# B&R Automation Studio project mappView-Backup
Automation Studio 4.5.4.123 SP

## Configuration X20CPU

### Task classes (Cpu.sw)
```
Cyclic#7:
  Test <- Test.prg
Cyclic#8:
  mappBackup <- mappBackup.mappBackup.prg
  UsbDevice <- USBdevice.UsbDevice.prg
  NetDevice <- NETdevice.NetDevice.prg
Binaries: udbdef, mvLoader, TCData, arsvcreg, sysconf, ashwd, ashwac, asfw, iomap, Role, User, arconfig, OpcUaMap, Config
Libraries: FileIO, runtime, AsBrStr, AsUSB, standard, sys_lib, MpBackup, MpBase, IecCheck, AsBrWStr, astime, asieccon, brsystem, arproject, asarcfg
```

### Hardware
```
X20CP1583 : X20CP1583 v1.5.0.0
  Connector IF2:
    ActivateDevice = 1
  ConfigurationID = Tmp_Backup
  UserPartitionSize = 32
  VolatileGlobalPvSize = 200000
  Cyclic8Stack = 20000
  FileDevice1
  FileDeviceName1 = USER_DEVICE
  FileDevicePath1 = F:/
  FtpUser1
  FtpUsername1 = br
  FtpUserPassword1 = B9fKGuUbjkGCgEptWUpgQ1eJbLeEvMYqPBCteWUIcCw=
  FtpUserSalt1 = wEo/3/qm
  FTPAccessRight1 = 0
  ActivateOpcUa = 1
  OpcUaInformationModels_PV_Version = 1
```

### Config.mpbackupcore - X20CP1583/mappServices/Config.mpbackupcore
```
Element gBackupCore (Type=mpbackupcore)
  Backup:
    AutomaticUpdate = Notify
      DeviceName = USBdevice
```

## Logical view

Binary libraries used (declarations not repeated): operator, runtime, astime, AsIecCon, FileIO, AsBrStr, AsUSB, standard, sys_lib, MpBackup 5.07.1, MpBase, IecCheck, AsBrWStr

### Package Logical/Libraries - Global libraries

- Visualisation Logical/mappView (not shown)

### BackupTypes.typ
```iecst
(*------------------------------------------------------------------------------------------------------------------------------------------------------------------------------------------------------------------------*)
(*Global enumerations*)

TYPE
	bacSTATE :
		( (*Backup managment state machine*)
		BAC_STARTUP,
		BAC_WAIT,
		BAC_CORE,
		BAC_FINISH,
		BAC_GENERATE_NAME,
		BAC_READ_DIR_0,
		BAC_READ_DIR_1,
		BAC_READ_DIR_2,
		BAC_READ_DIR_3,
		BAC_READ_DIR_4,
		BAC_DIR_DELETE,
		BAC_DIR_CREATE,
		BAC_ERROR
		);
END_TYPE

(*------------------------------------------------------------------------------------------------------------------------------------------------------------------------------------------------------------------------*)
(*Global structure*)

TYPE
	bacMAIN : 	STRUCT  (*Backup managment main structure*)
		CMD : bacCMD; (* Command structure *)
		PAR : bacPAR; (* Parameter structure *)
		DAT : bacDAT; (*Data structure*)
		VIS : bacVIS; (*Visualization structure*)
		ERR : bacERR; (* Error structure *)
	END_STRUCT;
	bacCMD : 	STRUCT  (*Backup managment command structure*)
		Backup : BOOL; (*Create a new backup*)
		Restore : BOOL; (*Restore selected backup*)
		Delete : BOOL; (*Delete the selected backaup*)
		GenerateName : BOOL; (*Generate backup name from default name and date*)
		RefreshInfo : BOOL; (*Refresh information for selected backup*)
		RefreshDirectory : BOOL; (*Refresh backup directory names*)
		ErrorReset : BOOL; (*Reset pending errors*)
	END_STRUCT;
	bacPAR : 	STRUCT  (*Backup managment parameter structure*)
		BackupName : STRING[BACKUP_NAME_LENGTH] := 'MyBackup'; (*Name of the variable where the data is stored*)
		DefaultName : STRING[BACKUP_NAME_LENGTH] := 'MyBackup'; (*Name of the variable where the data is stored*)
		DeviceName : STRING[BACKUP_NAME_LENGTH] := 'USB_DEVICE'; (*Device name where the bacipes are stored*)
		UniqueName : STRING[BACKUP_NAME_LENGTH] := 'RestoreInProcessPLC1'; (*Unique name for this PLC to identify if restore was completed*)
		DeviceList : ARRAY[0..4]OF STRING[40]; (*List of all devices*)
		VisuSlotID : USINT; (*ID for connected web connection*)
		ShowMessageBoxOK : BOOL := TRUE;
		ShowMessageBoxError : BOOL := TRUE;
		MpLink : MpComIdentType; (*MpLink from mappBackup*)
	END_STRUCT;
	bacDAT : 	STRUCT  (*Backup managment data structure*)
		CurrentID : STRING[255];
		CurrentVersion : STRING[64];
		RequestedName : STRING[255];
		RequestedID : STRING[255];
		RequestedVersion : STRING[64];
		LastName : STRING[255];
		LastDate : DATE_AND_TIME;
		LastType : MpBackupGenerationTypeEnum;
		BackupNames : ARRAY[0..BACKUP_LIST_NUM]OF STRING[BACKUP_NAME_LENGTH];
		BackupNum : USINT;
		Status : WSTRING[200]; (*Shows the result of the last command*)
	END_STRUCT;
	bacVIS : 	STRUCT  (*Backup managment visualization structure*)
		DeviceList : ARRAY[0..4]OF STRING[80]; (* Device name *)
		BackupNames : ARRAY[0..BACKUP_LIST_NUM]OF STRING[BACKUP_VIS_LENGTH];
		EnableCommand : BOOL;
		EnableDelete : BOOL;
		ShowMessageBoxOK : BOOL;
		ShowMessageBoxError : BOOL;
	END_STRUCT;
	bacERR : 	STRUCT  (*Backup managment error structure*)
		Text : WSTRING[200]; (* Error text *)
		No : DINT; (* Error number *)
		State : bacSTATE; (* Error step *)
	END_STRUCT;
END_TYPE
```

### BackupVariables.var
```iecst
VAR CONSTANT
	BACKUP_DEVICE_LIST : ARRAY[0..4] OF STRING[40] := ['USB_DEVICE','NET_DEVICE',3('')]; (*List of predefined devices *)
	BACKUP_LIST_NUM : UINT := 20; (*Maximum number of backups*)
	BACKUP_NAME_LENGTH : UINT := 100; (*Maximum length for a backup name*)
	BACKUP_VIS_LENGTH : UINT := 300; (*Make this BACKUP_NAME_LENGTH  x3*)
END_VAR
VAR
	BACKUP_DIRECTORY : STRING[200]; (*Directory for backups*)
	Backup_01 : bacMAIN; (*Backup management main structure*)
END_VAR
```

### Program Logical/mappBackup/mappBackup (IEC) - Sample for all AsUSB-Library-Functions

#### Backup.st - Cyclic code
```iecst
// ----------------------------------------------------------------------------------------
//	Function:	Software management for B&R PLCs
//  Version:	0.1
//	Changed:	11.11.2019
//	Error numbers:
//	50000		Backup name is empty
//	50001		Device name is empty
//	50010		Maximum number of backup names reached
//	50011		Backup name length exceeds maximum size
//	50020		Backup name already exists
// ----------------------------------------------------------------------------------------

PROGRAM _INIT
	// ----------------------------------------------------------------------------------------
	Backup_01.PAR.MpLink := gBackupCore;				// Link to mappBackup configuration

	// ----------------------------------------------------------------------------------------
	brsmemcpy(ADR(Backup_01.PAR.DeviceList), ADR(BACKUP_DEVICE_LIST), SIZEOF(BACKUP_DEVICE_LIST));
	Backup_01.DAT.Status := "Waiting...";

	MpBackupCore_0.MpLink := ADR(Backup_01.PAR.MpLink);
	MpBackupCore_0.Name := ADR(BackupName);
	MpBackupCore_0.DeviceName := ADR(DeviceName);

END_PROGRAM

PROGRAM _CYCLIC
	// --------------------------------------------------------------------------------------------------------------------
	// Cyclic function call
	MpBackupCore_0.Enable := 1;
	MpBackupCore_0();

	// ------------------------------------------------------------------------------------------------
	// Generate device name list
	brsmemset(ADR(Backup_01.VIS.DeviceList), 0, SIZEOF(Backup_01.VIS.DeviceList));
	FOR idx := 0 TO SIZEOF(Backup_01.VIS.DeviceList)/SIZEOF(Backup_01.VIS.DeviceList[0]) - 1 DO
		IF (Backup_01.PAR.DeviceList[idx] <> '') THEN
			String2DataProvider(ADR(Backup_01.PAR.DeviceList[idx]), ADR(Backup_01.VIS.DeviceList[idx]));
		END_IF
	END_FOR;

	// ------------------------------------------------------------------------------------------------
	// Generate backup name list
	brsmemset(ADR(Backup_01.VIS.BackupNames), 0, SIZEOF(Backup_01.VIS.BackupNames));
	IF(Backup_01.DAT.BackupNum > 0) THEN
		FOR idx := 0 TO Backup_01.DAT.BackupNum - 1 DO
			IF (Backup_01.DAT.BackupNames[idx] <> '') THEN
				String2DataProvider(ADR(Backup_01.DAT.BackupNames[idx]), ADR(Backup_01.VIS.BackupNames[idx]));
			END_IF
		END_FOR;
	END_IF

	// ------------------------------------------------------------------------------------------------
	// Enable/Disable visualization elements
	IF(bac_state <> BAC_WAIT) THEN
		Backup_01.VIS.EnableCommand := FALSE;
	ELSE
		Backup_01.VIS.EnableCommand := TRUE;
	END_IF
	IF(Backup_01.DAT.BackupNum = 0) THEN
		Backup_01.VIS.EnableDelete := FALSE;
	ELSE
		Backup_01.VIS.EnableDelete := TRUE;
	END_IF

	//**************************************************************************************************
	// Backup managment state machine
	//**************************************************************************************************
	CASE bac_state OF
		//**********************************************************************************************
		// Wait for USB and network connection to startup
		//**********************************************************************************************
		BAC_STARTUP:
			Backup_01.DAT.Status := "Waiting for USB and network connections to startup";
			StartupDelay(IN := 1, PT := DELAY_STARTUP);
			IF (StartupDelay.Q) THEN
				bac_state := BAC_WAIT;
			END_IF
		//**********************************************************************************************
		// Wait for command
		//**********************************************************************************************
		BAC_WAIT:
			// ----------------------------------------------------------------------------------------
			// Make sure device name is not empty
			IF ((Backup_01.CMD.Backup = TRUE OR Backup_01.CMD.Restore = TRUE OR Backup_01.CMD.Delete = TRUE OR Backup_01.CMD.RefreshDirectory = TRUE OR Backup_01.CMD.RefreshInfo = TRUE) AND Backup_01.PAR.DeviceName = '') THEN
				bac_state := CreateError(ADR(Backup_01), ERR_BAC_NAME_IS_EMPTY, "Device name is empty", bac_state);
				RETURN;
			ELSE
				// Freeze device name
				DeviceName := Backup_01.PAR.DeviceName;
			END_IF

			// ----------------------------------------------------------------------------------------
			// Make sure backup name is not empty
			IF ((Backup_01.CMD.Backup = TRUE OR Backup_01.CMD.Restore = TRUE OR Backup_01.CMD.Delete = TRUE OR Backup_01.CMD.RefreshInfo = TRUE) AND Backup_01.PAR.BackupName = '') THEN
				bac_state := CreateError(ADR(Backup_01), ERR_BAC_DEVICE_IS_EMPTY, "Backup name is empty", bac_state);
				RETURN;
			ELSE
				// Freeze backup name
				BackupName := Backup_01.PAR.BackupName;
			END_IF

			// ------------------------------------------------------------------------------------------------
			// Track device name change
			IF (brsstrcmp(ADR(DeviceNameOld), ADR(DeviceName)) <> 0) THEN
				Backup_01.CMD.RefreshDirectory	:= 1;
			END_IF
			DeviceNameOld := DeviceName;

			// ----------------------------------------------------------------------------------------
			// Command restore backup
			IF (Backup_01.CMD.Restore = TRUE) THEN
				// Show current state
				tmpWStr1 := "Restoring backup...";
				bac_state := BAC_DIR_CREATE;
			// ----------------------------------------------------------------------------------------
			// Command create backup
			ELSIF (Backup_01.CMD.Backup = TRUE) THEN
				// Make sure that backup name does not already exist
				IF(Backup_01.DAT.BackupNum > 0) THEN
					FOR idx:=0 TO Backup_01.DAT.BackupNum - 1 DO
						IF(brsstrcmp(ADR(BackupName), ADR(Backup_01.DAT.BackupNames[idx])) = 0) THEN
							bac_state := CreateError(ADR(Backup_01), ERR_BAC_NAME_EXISTS, "Backup name already exists", bac_state);
							RETURN;
						END_IF
					END_FOR;
				END_IF

				// Show current state
				tmpWStr1 := "Creating backup...";
				bac_state := BAC_CORE;
			// ----------------------------------------------------------------------------------------
			// Command delete backup
			ELSIF (Backup_01.CMD.Delete = TRUE) THEN
				// Show current state
				tmpWStr1 := "Deleting backup...";
				bac_state := BAC_DIR_DELETE;
			// ----------------------------------------------------------------------------------------
			// Command refresh backup information
			ELSIF (Backup_01.CMD.RefreshInfo = TRUE) THEN
				// Show current state
				tmpWStr1 := "Refreshing backup information...";
				bac_state := BAC_CORE;
			// ----------------------------------------------------------------------------------------
			// Command refresh device information
			ELSIF (Backup_01.CMD.RefreshDirectory = TRUE) THEN
				// Show current state
				tmpWStr1 := "Refreshing direct ory information...";
				DeviceIdx := 0;
				found_restore_dir := FALSE;
				DeviceName := Backup_01.PAR.DeviceName;
				bac_state := BAC_READ_DIR_0;
			// ----------------------------------------------------------------------------------------
			// Command generate backup name
			ELSIF (Backup_01.CMD.GenerateName = TRUE) THEN
				// Generate backup name
				bac_state := BAC_GENERATE_NAME;
			// ----------------------------------------------------------------------------------------
			// Command reset error
			ELSIF (Backup_01.CMD.ErrorReset = TRUE) THEN
				// Generate backup name
				bac_state := BAC_ERROR;
			END_IF

			animation := 0;
			MpBackupCore_0.ErrorReset := FALSE;
		//**********************************************************************************************
		// Generate backup name
		//**********************************************************************************************
		BAC_GENERATE_NAME:
			// Generate backup name using default name and date
			Backup_01.PAR.BackupName := Backup_01.PAR.DefaultName;
			RTC_gettime(ADR(rtc_gettime));
			brsstrcat(ADR(Backup_01.PAR.BackupName), ADR('_D'));
			IF(rtc_gettime.day < 10) THEN
				brsstrcat(ADR(Backup_01.PAR.BackupName), ADR('0'));
			END_IF
			brsitoa(rtc_gettime.day, ADR(tmpStr1));
			brsstrcat(ADR(Backup_01.PAR.BackupName), ADR(tmpStr1));
			brsitoa(rtc_gettime.day, ADR(tmpStr1));
			brsstrcat(ADR(Backup_01.PAR.BackupName), ADR('_M'));
			IF(rtc_gettime.month < 10) THEN
				brsstrcat(ADR(Backup_01.PAR.BackupName), ADR('0'));
			END_IF
			brsitoa(rtc_gettime.month, ADR(tmpStr1));
			brsstrcat(ADR(Backup_01.PAR.BackupName), ADR(tmpStr1));
			brsstrcat(ADR(Backup_01.PAR.BackupName), ADR('_Y'));
			brsitoa(rtc_gettime.year, ADR(tmpStr1));
			brsstrcat(ADR(Backup_01.PAR.BackupName), ADR(tmpStr1));
			brsstrcat(ADR(Backup_01.PAR.BackupName), ADR('_h'));
			IF(rtc_gettime.hour < 10) THEN
				brsstrcat(ADR(Backup_01.PAR.BackupName), ADR('0'));
			END_IF
			brsitoa(rtc_gettime.hour, ADR(tmpStr1));
			brsstrcat(ADR(Backup_01.PAR.BackupName), ADR(tmpStr1));
			brsstrcat(ADR(Backup_01.PAR.BackupName), ADR('_m'));
			IF(rtc_gettime.minute < 10) THEN
				brsstrcat(ADR(Backup_01.PAR.BackupName), ADR('0'));
			END_IF
			brsitoa(rtc_gettime.minute, ADR(tmpStr1));
			brsstrcat(ADR(Backup_01.PAR.BackupName), ADR(tmpStr1));
			brsstrcat(ADR(Backup_01.PAR.BackupName), ADR('_s'));
			IF(rtc_gettime.second < 10) THEN
				brsstrcat(ADR(Backup_01.PAR.BackupName), ADR('0'));
			END_IF
			brsitoa(rtc_gettime.second, ADR(tmpStr1));
			brsstrcat(ADR(Backup_01.PAR.BackupName), ADR(tmpStr1));

			Backup_01.CMD.GenerateName := FALSE;
			bac_state := BAC_WAIT;
		// --------------------------------------------------------------------------------------------------------------------
		// Core function call
		// --------------------------------------------------------------------------------------------------------------------
		BAC_CORE:
			// ------------------------------------------------------------------------------------------------
			// Main backup function call
			animation := WorkingStatus(ADR(Backup_01), ADR(tmpWStr1), animation);

			// ----------------------------------------------------------------------------------------
			// OK
			IF (MpBackupCore_0.CommandDone AND NOT MpBackupCore_0.Error) THEN
				IF(Backup_01.CMD.RefreshInfo OR Backup_01.CMD.Restore) THEN
					bac_state := BAC_FINISH;
				ELSE
					bac_state := BAC_READ_DIR_0;
				END_IF
				// ----------------------------------------------------------------------------------------
			// Error
			ELSIF (MpBackupCore_0.Error) THEN
				// ----------------------------------------------------------------------------------------
				// Generate error message depending on initial command
				IF (Backup_01.CMD.Backup) THEN
					IF(MpBackupCore_0.StatusID =  mpBACKUP_ERR_CREATE_FAILED) THEN
						tmpWStr1 := "Backup name already exists";
					ELSE
						tmpWStr1 := "Error trying to backup data";
					END_IF
				ELSIF (Backup_01.CMD.Restore) THEN
					IF(MpBackupCore_0.StatusID =  mpBACKUP_ERR_INSTALL_FAILED) THEN
						tmpWStr1 := "Can not find backup name";
					ELSE
						tmpWStr1 := "Error trying to restore data";
					END_IF
				ELSIF (Backup_01.CMD.RefreshInfo) THEN
					IF(MpBackupCore_0.StatusID =  mpBACKUP_ERR_REQUEST_INFO_FAILED) THEN
						bac_state := BAC_FINISH;
						RETURN;
					ELSE
						tmpWStr1 := "Error trying to refresh backup information";
					END_IF
				END_IF
				bac_state := CreateError(ADR(Backup_01), MpBackupCore_0.StatusID, tmpWStr1, bac_state);
			END_IF
		//**********************************************************************************************
		// Finish command
		//**********************************************************************************************
		BAC_FINISH:
			// ----------------------------------------------------------------------------------------
			// Comand backup
			IF (Backup_01.CMD.Backup) THEN
				// Reset command, set status and show message box
				Backup_01.DAT.Status := "Backup completed";
				IF(Backup_01.PAR.ShowMessageBoxOK) THEN
					Backup_01.VIS.ShowMessageBoxOK := TRUE;
				END_IF
			// ----------------------------------------------------------------------------------------
			// Comand restore
			ELSIF (Backup_01.CMD.Restore) THEN
				// Reset command, set status, return to wait state
				Backup_01.DAT.Status := "Restore backup completed";
			// ----------------------------------------------------------------------------------------
			// Comand delete
			ELSIF (Backup_01.CMD.Delete) THEN
				// Reset command, set status, return to wait state
				Backup_01.DAT.Status := "Deleted backup";
				IF(Backup_01.PAR.ShowMessageBoxOK) THEN
					Backup_01.VIS.ShowMessageBoxOK := TRUE;
				END_IF
			// ----------------------------------------------------------------------------------------
			// Comand refresh backup names
			ELSIF (Backup_01.CMD.RefreshDirectory) THEN
				// Show error message if there are oversized items
				IF(found_restore_dir) THEN
					// Reset command, set status, return to wait state
					found_restore_dir := FALSE;
					Backup_01.DAT.Status := "Restore backup complete";
					IF(Backup_01.PAR.ShowMessageBoxOK) THEN
						Backup_01.VIS.ShowMessageBoxOK := TRUE;
					END_IF
				ELSE
					Backup_01.DAT.Status := "Refreshed backup names";
				END_IF
			// ----------------------------------------------------------------------------------------
			// Comand refresh backup information
			ELSIF (Backup_01.CMD.RefreshInfo) THEN
				// Directory does not contain a PLC backup
				IF(MpBackupCore_0.StatusID =  mpBACKUP_ERR_REQUEST_INFO_FAILED) THEN
					Backup_01.DAT.Status := "Can not find directory or backup information";
				ELSE
					Backup_01.DAT.Status := "Refreshed backup information";
				END_IF
			END_IF
			// Set status, return to wait state
			brsmemset(ADR(Backup_01.CMD), 0, SIZEOF(Backup_01.CMD));
			MpBackupCore_0.ErrorReset := TRUE;
			MpBackupCore_0();
			MpBackupCore_0.ErrorReset := FALSE;
			bac_state := BAC_WAIT;
		//**********************************************************************************************
		// Read directory information
		//**********************************************************************************************
		BAC_READ_DIR_0:
			// Show current state
			animation := WorkingStatus(ADR(Backup_01), ADR(tmpWStr1), animation);
			// Clear all entrys, reset mappBackup function block
			brsmemset(ADR(Backup_01.DAT), 0, SIZEOF(Backup_01.DAT));
			Backup_01.DAT.BackupNum := 0;
			has_oversized_items := FALSE;

			// ----------------------------------------------------------------------------------------
			// Reset mappBackup function block
			MpBackupCore_0.Enable := 0;
			MpBackupCore_0();
			// ----------------------------------------------------------------------------------------
			// Set values and get device dir
			DInfo.enable 	:= 1;
			DInfo.pDevice	:= ADR(DeviceName);
			DInfo();

			// ----------------------------------------------------------------------------------------
			// OK
			IF (DInfo.status = OK) THEN
				first_boot := FALSE;
				bac_state := BAC_READ_DIR_1;
			ELSIF (DInfo.status = fiERR_DEVICE_MANAGER) THEN
				// On first boot skip devices that are not available
				IF (first_boot) THEN
					DeviceIdx := DeviceIdx + 1;
					IF(Backup_01.PAR.DeviceList[DeviceIdx] <> '') THEN
						brsstrcpy(ADR(DeviceName), ADR(Backup_01.PAR.DeviceList[DeviceIdx]));
						brsstrcpy(ADR(DeviceNameOld), ADR(Backup_01.PAR.DeviceList[DeviceIdx]));
						brsstrcpy(ADR(Backup_01.PAR.DeviceName), ADR(Backup_01.PAR.DeviceList[DeviceIdx]));
					ELSE
						// Set status, return to wait state
						brsmemset(ADR(Backup_01.CMD), 0, SIZEOF(Backup_01.CMD));
						first_boot := FALSE;
						bac_state := BAC_WAIT;
					END_IF
				// Create error message when file device is not available
				ELSE
					tmpWStr1 := "File device ";
					brwcsconv(ADR(tmpWStr2), ADR(DeviceName), brwU8toUC);
					brwcscat(ADR(tmpWStr1), ADR(tmpWStr2));
					brwcscat(ADR(tmpWStr1), ADR(" is unavailable"));
					bac_state := CreateError(ADR(Backup_01), DInfo.status, tmpWStr1, bac_state);
				END_IF
			// Error
			ELSIF (DInfo.status <> ERR_FUB_BUSY) THEN
				first_boot := FALSE;
				bac_state := CreateError(ADR(Backup_01), DInfo.status, "Error dir info", bac_state);
			END_IF
		//**********************************************************************************************
		// Open directory
		//**********************************************************************************************
		BAC_READ_DIR_1:
			// Show current state
			animation := WorkingStatus(ADR(Backup_01), ADR(tmpWStr1), animation);

			DOpen.enable 	:= 1;
			DOpen.pDevice	:= ADR(DeviceName);
			DOpen.pName 	:= ADR(BACKUP_DIRECTORY);
			DOpen();

			// ----------------------------------------------------------------------------------------
			// OK
			IF (DOpen.status = OK) THEN
				bac_state := BAC_READ_DIR_2;
				// Error
			ELSIF (DOpen.status <> ERR_FUB_BUSY) THEN
				bac_state := CreateError(ADR(Backup_01), DOpen.status, "Error dir open", bac_state);
			END_IF;
		//**********************************************************************************************
		// Read file directory information
		//**********************************************************************************************
		BAC_READ_DIR_2:
			// Show current state
			animation := WorkingStatus(ADR(Backup_01), ADR(tmpWStr1), animation);

			DRead.enable 	:= 1;
			DRead.ident		:= DOpen.ident;
			DRead.pData 	:= ADR(lDirReadData);
			DRead.data_len 	:= SIZEOF(lDirReadData);
			DRead();

			// ----------------------------------------------------------------------------------------
			// OK
			IF (DRead.status = OK AND lDirReadData.Mode = fiDIRECTORY AND brsstrcmp(ADR(lDirReadData.Filename), ADR('.')) <> 0 AND brsstrcmp(ADR(lDirReadData.Filename), ADR('..')) <> 0 AND brsstrcmp(ADR(lDirReadData.Filename), ADR('System Volume Information')) <> 0) THEN
				// Make sure file name does not exceed maximum string size
				IF (brsstrlen(ADR(lDirReadData.Filename)) < BACKUP_NAME_LENGTH) THEN
					// Copy dir info to string
					brsmemset(ADR(tmpStr1), 0, SIZEOF(tmpStr1));
					brsstrcpy(ADR(tmpStr1), ADR(lDirReadData.Filename));
					// Found restore directory
					IF(brsstrcmp(ADR(Backup_01.PAR.UniqueName), ADR(tmpStr1)) = 0) THEN
						found_restore_dir := TRUE;
					ELSE
						// ------------------------------------------------------------------------------------
						// Verify that we still have space in list
						IF (Backup_01.DAT.BackupNum <= BACKUP_LIST_NUM) THEN
							InsertRecName(ADR(Backup_01), tmpStr1);
							// Error
						ELSE
							bac_state := CreateError(ADR(Backup_01), ERR_BAC_MAX_NUM, "Maximum number of backups reached", bac_state);
						END_IF
					END_IF
				ELSE
					has_oversized_items := TRUE;
				END_IF
			// Last entry reached
			ELSIF (DRead.status = fiERR_NO_MORE_ENTRIES) THEN
				bac_state := BAC_READ_DIR_3;
			// Error
			ELSIF (DRead.status <> ERR_FUB_BUSY AND DRead.status <> OK) THEN
				bac_state := CreateError(ADR(Backup_01), DRead.status, "Error backup list read", bac_state);
			END_IF
		//**********************************************************************************************
		// Close directory information
		//**********************************************************************************************
		BAC_READ_DIR_3:
			// Show current state
			animation := WorkingStatus(ADR(Backup_01), ADR(tmpWStr1), animation);

			DClose.enable 	:= 1;
			DClose.ident	:= DOpen.ident;
			DClose();

			// ----------------------------------------------------------------------------------------
			// OK
			IF (DClose.status = OK) THEN
				// Delete restore flag directory
				IF(found_restore_dir) THEN
					BackupName := Backup_01.PAR.UniqueName;
					bac_state := BAC_DIR_DELETE;
				// Finish directory reading
				ELSE
					bac_state := BAC_READ_DIR_4;
				END_IF
			// Error
			ELSIF (DClose.status <> ERR_FUB_BUSY) THEN
				bac_state := CreateError(ADR(Backup_01), DClose.status, "Error dir close", bac_state);
			END_IF
		//**********************************************************************************************
		// Finish directory information
		//**********************************************************************************************
		BAC_READ_DIR_4:
			// Show error message if there are oversized items
			IF(has_oversized_items) THEN
				bac_state := CreateError(ADR(Backup_01), ERR_BAC_NAME_LENGTH, "One or more backup names exceeds maximum length", bac_state);
			ELSE
				// Get information from first entry
				IF(Backup_01.DAT.BackupNum > 0) THEN
					BackupName := Backup_01.DAT.BackupNames[0];
					Backup_01.CMD.RefreshInfo := TRUE;
					bac_state := BAC_CORE;
				ELSE
					bac_state := BAC_FINISH;
				END_IF
			END_IF
		//**********************************************************************************************
		// Delete selected directory
		//**********************************************************************************************
		BAC_DIR_DELETE:
			// Show current state
			animation := WorkingStatus(ADR(Backup_01), ADR("Deleting backup..."), animation);

			// ----------------------------------------------------------------------------------------
			// Initialize directory delete structure
			DDelete.enable	:= 1;
			DDelete.pDevice := ADR(DeviceName);
			DDelete.pName 	:= ADR(BackupName);
			DDelete();

			// ----------------------------------------------------------------------------------------
			// OK
			IF (DDelete.status = OK) THEN
				// Deleted restore directory
				IF(found_restore_dir) THEN
					bac_state := BAC_READ_DIR_4;
				// Deleted standard backup directory
				ELSE
					// Show status and return to wait state
					Backup_01.DAT.Status := "Deleted backup";
					bac_state := BAC_READ_DIR_0;
				END_IF
			// Error
			ELSIF (DDelete.status <> ERR_FUB_BUSY) THEN
				IF(DDelete.status = fiERR_DIR_NOT_EXIST) THEN
					bac_state := CreateError(ADR(Backup_01), DDelete.status, "Can not find backup directory", bac_state);
				ELSE
					bac_state := CreateError(ADR(Backup_01), DDelete.status, "Error deleting backup", bac_state);
				END_IF
			END_IF
		//**********************************************************************************************
		// Create selected directory
		//**********************************************************************************************
		BAC_DIR_CREATE:
			// Show current state
			animation := WorkingStatus(ADR(Backup_01), ADR(tmpWStr1), animation);

			// ----------------------------------------------------------------------------------------
			// Initialize directory delete structure
			DCreate.enable	:= 1;
			DCreate.pDevice := ADR(DeviceName);
			DCreate.pName 	:= ADR(Backup_01.PAR.UniqueName);
			DCreate();

			// ----------------------------------------------------------------------------------------
			// OK
			IF (DCreate.status = OK OR DCreate.status = fiERR_DIR_ALREADY_EXIST) THEN
				// Start restoring backup
				bac_state := BAC_CORE;
			// Error
			ELSIF (DCreate.status <> ERR_FUB_BUSY) THEN
				bac_state := CreateError(ADR(Backup_01), DCreate.status, "Could not create restore flag directory", bac_state);
			END_IF
		// --------------------------------------------------------------------------------------------------------------------
		// Error
		// --------------------------------------------------------------------------------------------------------------------
		BAC_ERROR:
			Backup_01.DAT.Status := "Acknowledge error to trigger new command";

			// Make sure we dont exceed maximum number of web clients
			IF(Backup_01.PAR.ShowMessageBoxError) THEN
				Backup_01.VIS.ShowMessageBoxError := TRUE;
			END_IF
			// --------------------------------------------------------------------------------------------------------------------
			// Return to idle state
			IF (Backup_01.CMD.ErrorReset) THEN
				// Reset function blocks
				MpBackupCore_0.ErrorReset := TRUE;
				MpBackupCore_0();
				MpBackupCore_0.ErrorReset := FALSE;

				// Reset error structure
				brsmemset(ADR(Backup_01.ERR), 0, SIZEOF(Backup_01.ERR));
				Backup_01.DAT.Status := "";
				Backup_01.VIS.ShowMessageBoxError := FALSE;
				bac_state := BAC_WAIT;
			END_IF;
			brsmemset(ADR(Backup_01.CMD), 0, SIZEOF(Backup_01.CMD));
	END_CASE

	// --------------------------------------------------------------------------------------------------------------------
	// Cyclic function call
	MpBackupCore_0.Enable := 1;
	MpBackupCore_0.Create := Backup_01.CMD.Backup;
	MpBackupCore_0.Install := Backup_01.CMD.Restore;
	MpBackupCore_0.RequestInfo := Backup_01.CMD.RefreshInfo;
	MpBackupCore_0();

	Backup_01.DAT.CurrentID := MpBackupCore_0.Info.Project.Current.ConfigurationID;
	Backup_01.DAT.CurrentVersion := MpBackupCore_0.Info.Project.Current.ConfigurationVersion;
	Backup_01.DAT.RequestedName := MpBackupCore_0.Info.Project.Requested.Name;
	Backup_01.DAT.RequestedID := MpBackupCore_0.Info.Project.Requested.ConfigurationID;
	Backup_01.DAT.RequestedVersion := MpBackupCore_0.Info.Project.Requested.ConfigurationVersion;
	Backup_01.DAT.LastName := MpBackupCore_0.Info.LastBackup.Name;
	Backup_01.DAT.LastDate := MpBackupCore_0.Info.LastBackup.DateTime;
	Backup_01.DAT.LastType := MpBackupCore_0.Info.LastBackup.GenerationType;

END_PROGRAM

PROGRAM _EXIT
	MpBackupCore_0.Enable := 0;
	MpBackupCore_0();
END_PROGRAM
```

#### Backup.var - Data for read_data Task
```iecst
(*------------------------------------------------------------------------------------------------------------------------------------------------------------------------------------------------------------------------*)
(*Local constants*)
VAR CONSTANT
	OK : USINT := 0; (*Constant for status OK *)
END_VAR
VAR
	DELAY_STARTUP : UINT := 1000; (*Delay startup to give USB and network connections time to start up*)
END_VAR
(*----------------------------------------------------------------------------------------------------------------------------------------------------------------------------------------------------------------------------------------------------------------------*)
(*Local variables*)
VAR
	bac_state : bacSTATE := BAC_STARTUP; (*Main step index *)
	first_boot : BOOL := TRUE; (*Flag for first boot up, run some special code*)
	animation : UDINT := 0; (*Animation for working status	*)
	tmpWStr1 : WSTRING[200]; (*Temporary unicode string variable *)
	tmpWStr2 : WSTRING[200]; (*Temporary unicode string variable *)
	tmpStr1 : STRING[100]; (*Temporary string variable *)
	BackupName : STRING[BACKUP_NAME_LENGTH]; (*Local backup name*)
	DeviceNameOld : STRING[100]; (*Local device name*)
	DeviceName : STRING[100]; (*Local device name*)
	DeviceIdx : USINT;
	idx : UINT; (*Counter variable*)
	rtc_gettime : RTCtime_typ; (*Time and date*)
	lDirReadData : fiDIR_READ_EX_DATA; (*File and directory information*)
	has_oversized_items : BOOL; (*Flag for oversized backup names*)
	found_restore_dir : BOOL; (*Flag for directory for the restpre process*)
END_VAR
(*----------------------------------------------------------------------------------------------------------------------------------------------------------------------------------------------------------------------------------------------------------------------*)
(*Local functions*)
VAR
	MpBackupCore_0 : MpBackupCore; (*mappBackup function block*)
	DInfo : DirInfo; (*Directory information*)
	DOpen : DirOpen; (*Start reading directories*)
	DRead : DirReadEx; (*Read directories*)
	DClose : DirClose; (*Finish reading directories*)
	DDelete : DirDeleteEx; (*Delete directory*)
	DCreate : DirCreate; (*Finish reading directories*)
	StartupDelay : TON_10ms; (*Delay startup timer*)
END_VAR
(*----------------------------------------------------------------------------------------------------------------------------------------------------------------------------------------------------------------------------------------------------------------------*)
(*Local errors*)
VAR
	ERR_BAC_NAME_IS_EMPTY : DINT := 50000; (*Backup name is empty*)
	ERR_BAC_DEVICE_IS_EMPTY : DINT := 50001; (*Device name is empty*)
	ERR_BAC_MAX_NUM : DINT := 50010; (*Maximum number of backup names reached*)
	ERR_BAC_NAME_LENGTH : DINT := 50011; (*Backup name length exceeds maximum size*)
	ERR_BAC_NAME_EXISTS : DINT := 50020; (*Backup name already exists*)
END_VAR
```

#### LocalFunctions.fun
```iecst
FUNCTION String2DataProvider : BOOL
	VAR_INPUT
		SourceString : UDINT;
		TargetString : UDINT;
	END_VAR
END_FUNCTION

FUNCTION WorkingStatus : UDINT
	VAR_INPUT
		BACKUP : REFERENCE TO bacMAIN;
		str : UDINT;
		animation : UDINT;
	END_VAR
	VAR
		counter : UDINT;
		tmpStr : STRING[20];
		tmpWStr : WSTRING[20];
	END_VAR
END_FUNCTION

FUNCTION CreateError : bacSTATE
	VAR_INPUT
		BACKUP : REFERENCE TO bacMAIN;
		No : DINT;
		Text : WSTRING[200];
		State : bacSTATE;
	END_VAR
END_FUNCTION

FUNCTION InsertRecName : BOOL
	VAR_INPUT
		BAC : REFERENCE TO bacMAIN;
		new_name : STRING[BACKUP_NAME_LENGTH];
	END_VAR
	VAR
		idx : DINT;
		idy : DINT;
		lSort : DINT;
	END_VAR
END_FUNCTION
```

#### LocalFunctions.st
```iecst
//******************************************************************************************************
// Create mappView data provider string
//******************************************************************************************************
FUNCTION String2DataProvider
	brsstrcpy(TargetString, ADR('{"value":"'));
	brsstrcat(TargetString, SourceString);
	brsstrcat(TargetString, ADR('","text":"'));
	brsstrcat(TargetString, SourceString);
	brsstrcat(TargetString, ADR('"}'));
	String2DataProvider := TRUE;
END_FUNCTION

//******************************************************************************************************
// Create error
//******************************************************************************************************
FUNCTION CreateError
	BACKUP.ERR.No := No;
	BACKUP.ERR.State := State;
	BACKUP.ERR.Text := Text;
	CreateError := BAC_ERROR;
END_FUNCTION

//******************************************************************************************************
// Working status
//******************************************************************************************************
FUNCTION WorkingStatus
	animation := animation+1;

	// Get one second counter
	counter := animation;
	WHILE counter >= 100 DO
		counter := counter - 100;
	END_WHILE;

	IF (counter = 99) THEN
		counter := 0;
	END_IF

	// Add counter to output string
	brsmemset(ADR(BACKUP.DAT.Status), 0, SIZEOF(BACKUP.DAT.Status));
	brwcscpy(ADR(BACKUP.DAT.Status), str);
	brwcscat(ADR(BACKUP.DAT.Status), ADR(" "));
	brsitoa(animation/100, ADR(tmpStr));
	brwcsconv(ADR(tmpWStr), ADR(tmpStr), brwU8toUC);
	brwcscat(ADR(BACKUP.DAT.Status), ADR(tmpWStr));
	brwcscat(ADR(BACKUP.DAT.Status), ADR("s "));

	// Add rotating element to output string
	CASE(counter) OF
		0..24	: brwcscat(ADR(BACKUP.DAT.Status), ADR("/"));
		25..49	: brwcscat(ADR(BACKUP.DAT.Status), ADR("-"));
		50..74	: brwcscat(ADR(BACKUP.DAT.Status), ADR("\"));
		75..99	: brwcscat(ADR(BACKUP.DAT.Status), ADR("|"));
	END_CASE;
	WorkingStatus := animation;
END_FUNCTION

//******************************************************************************************************
// Fill in new directory name
//******************************************************************************************************
FUNCTION InsertRecName
	// Set up start values for iteration
	IF (BAC.DAT.BackupNum <> 0) THEN
		idy := BAC.DAT.BackupNum - 1;
	END_IF
	idx := idy;

	// Start iteration	search
	WHILE (idy > 1) DO
		// Check current entry
		lSort := brsstrcmp(ADR(new_name), ADR(BAC.DAT.BackupNames[idy]));
		// Solve new search range
		IF (idy MOD 2 = 0) THEN
			idy := idy / 2;
		ELSE
			idy := idy / 2 + 1;
		END_IF
		// New range is lower or higher than current
		IF (lSort > 0) THEN
			idx := idx + idy;
			IF (idx > UINT_TO_INT(BAC.DAT.BackupNum)) THEN
				idx := BAC.DAT.BackupNum;
			END_IF
		ELSE
			idx := idx - idy;
			IF (idx < 1) THEN
				idx := 1;
			END_IF
		END_IF
	END_WHILE;

	// New entry is this, next or previous
	lSort := brsstrcmp(ADR(new_name), ADR(BAC.DAT.BackupNames[idx]));
	IF (lSort > 0 AND idx <> UINT_TO_INT(BAC.DAT.BackupNum)) THEN
		idx := idx +1;
	ELSIF (idx > 0) THEN
		lSort := brsstrcmp(ADR(new_name), ADR(BAC.DAT.BackupNames[idx-1]));
		IF (lSort < 0) THEN
			idx := idx - 1;
		END_IF
	END_IF

	// Move all data entrys backwards and fill in new entry
	IF(idx < BACKUP_LIST_NUM) THEN
		brsmemmove(ADR(BAC.DAT.BackupNames[idx+1]),ADR(BAC.DAT.BackupNames[idx]), (BAC.DAT.BackupNum - idx) * SIZEOF(BAC.DAT.BackupNames[0]));
	END_IF
	brsstrcpy(ADR(BAC.DAT.BackupNames[idx]), ADR(new_name));
	BAC.DAT.BackupNum := BAC.DAT.BackupNum + 1;

	InsertRecName := TRUE;
END_FUNCTION
```

### changelog.txt
```
Version 0.2
- Added ping support for network share
- Fixed error message after network backup

Version 0.1
- First public release
```

### NetTypes.typ
```iecst
TYPE
	netSTATE :
		(
		NET_WAIT, (*Function step: Wait for starting the Function chain*)
		NET_LINK_DEVICE, (*Function step: Link file device*)
		NET_UNLINK_DEVICE, (*Function step: Unlink the File Device from specific path*)
		NET_ERROR (*Function step: Jump to this step in every case of Error occuring in the Function chain*)
		);
	netCMD : 	STRUCT
		connect : BOOL := TRUE; (*Connect to network share*)
		error_reset : BOOL; (*Reset error*)
	END_STRUCT;
	netPAR : 	STRUCT
		state_machine : netSTATE; (*State machine*)
		server_name : STRING[80]; (*Use server name*)
		server_ip : STRING[80] := '192.168.0.10'; (*or IP address*)
		server_port : STRING[80]; (*Uses default port when empty*)
		server_protocol : STRING[80] := 'cifs'; (*Type of network connection*)
		server_domain : STRING[80] := ''; (*Domain name*)
		server_share : STRING[80] := 'share'; (*Name of the shared folder*)
		user_name : STRING[80] := ''; (*User name*)
		user_password : STRING[80] := ''; (*User password*)
		enable_connect : BOOL; (*Enable button connect*)
		is_linked : BOOL; (*Network share is connected*)
	END_STRUCT;
	netERR : 	STRUCT
		no : UINT; (*Error number*)
		state : netSTATE;
		text : STRING[80]; (*Error text*)
		active : BOOL;
	END_STRUCT;
	netMAIN : 	STRUCT
		CMD : netCMD; (*Command structure*)
		PAR : netPAR; (*Parameter structure*)
		ERR : netERR; (*Error structure*)
	END_STRUCT;
END_TYPE
```

### changelog.txt
```
Version 0.2
- Fixed error message after network backup

Version 0.1
- First public release
```

### Program Logical/NETdevice/NetDevice

#### Variables.var
```iecst
(*----------------------------------------------------------------------------------------------------------------------------------------------------------------------------------------------------------------------------------------------------------------------*)
(*Local functions*)
VAR
	DevLink_0 : DevLink; (*Link network device*)
	DevUnlink_0 : DevUnlink; (*Unlink network device*)
	IcmpPing_0 : IcmpPing; (*Ping network share*)
END_VAR
(*----------------------------------------------------------------------------------------------------------------------------------------------------------------------------------------------------------------------------------------------------------------------*)
(*Local variables*)
VAR
	device_param : STRING[200]; (*Connection path of network device*)
	device_handle : UDINT;
END_VAR
```

#### Main.st
```iecst
PROGRAM _INIT
	(* Insert code here *)

END_PROGRAM

PROGRAM _CYCLIC
	// Try to ping network share if not connected
	IF((NET.PAR.server_ip <> '' OR NET.PAR.server_name <> '') AND NOT NET.PAR.is_linked) THEN
		IF(NET.PAR.server_ip <> '') THEN
			IcmpPing_0(enable := 1, pHost := ADR(NET.PAR.server_ip), timeout := 50);
		ELSE
			IcmpPing_0(enable := 1, pHost := ADR(NET.PAR.server_name), timeout := 50);
		END_IF
		IF(IcmpPing_0.status = ERR_OK) THEN
			NET.PAR.can_ping := TRUE;
		ELSIF(IcmpPing_0.status <> ERR_FUB_BUSY) THEN
			NET.PAR.can_ping := FALSE;
		END_IF
	END_IF

	CASE NET.PAR.state_machine OF
		// -----------------------------------------------------------------------------------------------------------
		// Wait state
		// -----------------------------------------------------------------------------------------------------------
		NET_WAIT:
			NET.PAR.enable_connect := TRUE;
			// --------------------------------------------------------------------------------------------------------------------
			// Connect to server
			IF(NET.CMD.connect) THEN
				IF(NET.PAR.is_linked) THEN
					DevUnlink_0.enable := 0;
					DevUnlink_0;
					IF (DevUnlink_0.status = ERR_FUB_ENABLE_FALSE) THEN
						NET.PAR.state_machine := NET_UNLINK_DEVICE;
					END_IF
				ELSE
					DevLink_0.enable := 0;
					DevLink_0;
					IF (DevLink_0.status = ERR_FUB_ENABLE_FALSE) THEN
						NET.PAR.state_machine := NET_LINK_DEVICE;
					END_IF
				END_IF
			END_IF
			// --------------------------------------------------------------------------------------------------------------------
			// Disconnect from server
			IF(NET.CMD.error_reset) THEN
				IF(NET.PAR.is_linked) THEN
					DevUnlink_0.enable := 0;
					DevUnlink_0;
					NET.PAR.state_machine := NET_UNLINK_DEVICE;
				ELSE
					NET.CMD.error_reset := FALSE;
				END_IF
				brsmemset(ADR(NET.ERR), 0, SIZEOF(NET.ERR));
			END_IF
		// -----------------------------------------------------------------------------------------------------------
		// Link device
		// -----------------------------------------------------------------------------------------------------------
		NET_LINK_DEVICE:
			// Create device string
			NET.PAR.enable_connect := FALSE;
			brsmemset(ADR(device_param), 0, SIZEOF(device_param));
			IF(brsstrcmp(ADR(NET.PAR.server_name), ADR('')) <> 0) THEN
				brsstrcat(ADR(device_param), ADR('/SNAME='));
				brsstrcat(ADR(device_param), ADR(NET.PAR.server_name));
				brsstrcat(ADR(device_param), ADR(' '));
			END_IF
			IF(brsstrcmp(ADR(NET.PAR.server_ip), ADR('')) <> 0) THEN
				brsstrcat(ADR(device_param), ADR('/SIP='));
				brsstrcat(ADR(device_param), ADR(NET.PAR.server_ip));
				brsstrcat(ADR(device_param), ADR(' '));
			END_IF
			IF(brsstrcmp(ADR(NET.PAR.server_protocol), ADR('')) <> 0) THEN
				brsstrcat(ADR(device_param), ADR('/PROTOCOL='));
				brsstrcat(ADR(device_param), ADR(NET.PAR.server_protocol));
				brsstrcat(ADR(device_param), ADR(' '));
			END_IF
			IF(brsstrcmp(ADR(NET.PAR.server_port), ADR('')) <> 0) THEN
				brsstrcat(ADR(device_param), ADR('/PORT='));
				brsstrcat(ADR(device_param), ADR(NET.PAR.server_port));
				brsstrcat(ADR(device_param), ADR(' '));
			END_IF
			IF(brsstrcmp(ADR(NET.PAR.server_domain), ADR('')) <> 0) THEN
				brsstrcat(ADR(device_param), ADR('/DOMAIN='));
				brsstrcat(ADR(device_param), ADR(NET.PAR.server_domain));
				brsstrcat(ADR(device_param), ADR(' '));
			END_IF
			IF(brsstrcmp(ADR(NET.PAR.server_share), ADR('')) <> 0) THEN
				brsstrcat(ADR(device_param), ADR('/SHARE='));
				brsstrcat(ADR(device_param), ADR(NET.PAR.server_share));
				brsstrcat(ADR(device_param), ADR(' '));
			END_IF
			IF(brsstrcmp(ADR(NET.PAR.user_name), ADR('')) <> 0) THEN
				brsstrcat(ADR(device_param), ADR('/USER='));
				brsstrcat(ADR(device_param), ADR(NET.PAR.user_name));
				brsstrcat(ADR(device_param), ADR(' '));
			END_IF
			IF(brsstrcmp(ADR(NET.PAR.user_password), ADR('')) <> 0) THEN
				brsstrcat(ADR(device_param), ADR('/PASSWORD='));
				brsstrcat(ADR(device_param), ADR(NET.PAR.user_password));
				brsstrcat(ADR(device_param), ADR(' '));
			END_IF

			// Link device
			DevLink_0.enable := 1;
			DevLink_0.pDevice := ADR('NET_DEVICE');
			DevLink_0.pParam := ADR(device_param);
			DevLink_0;

			// --------------------------------------------------------------------------------------------------------------------
			// Success
			IF DevLink_0.status = 0 THEN
				device_handle := DevLink_0.handle;
				NET.PAR.is_linked := TRUE;
				NET.CMD.connect := FALSE;
				NET.PAR.state_machine := NET_WAIT;
			// --------------------------------------------------------------------------------------------------------------------
			// Abort command
			ELSIF(NET.CMD.error_reset) THEN
				NET.CMD.error_reset := FALSE;
				NET.CMD.connect := FALSE;
				NET.PAR.state_machine := NET_WAIT;
				// Error
			ELSIF DevLink_0.status <> ERR_FUB_BUSY THEN
				NET.ERR.state := NET.PAR.state_machine;
				NET.ERR.no := DevLink_0.status;
				NET.ERR.text := 'error linking device';
				NET.PAR.state_machine := NET_ERROR;
			END_IF;
		// -----------------------------------------------------------------------------------------------------------
		// UnLink device
		// -----------------------------------------------------------------------------------------------------------
		NET_UNLINK_DEVICE:
			NET.PAR.enable_connect := FALSE;
			DevUnlink_0.enable := 1;
			DevUnlink_0.handle := device_handle;
			DevUnlink_0;

			// --------------------------------------------------------------------------------------------------------------------
			// Success
			IF DevUnlink_0.status = 0 THEN
				NET.PAR.is_linked := FALSE;
				IF(NET.CMD.connect) THEN
					DevLink_0.enable := 0;
					DevLink_0;
					NET.PAR.state_machine := NET_LINK_DEVICE;
				ELSE
					NET.CMD.error_reset := FALSE;
					NET.PAR.state_machine := NET_WAIT;
				END_IF
			// Error
			ELSIF DevUnlink_0.status <> ERR_FUB_BUSY THEN
				NET.CMD.error_reset := FALSE;
				NET.ERR.state := NET.PAR.state_machine;
				NET.ERR.no := DevUnlink_0.status;
				NET.ERR.text := 'error unlinking device';
				NET.PAR.state_machine := NET_ERROR;
			END_IF;
		// -----------------------------------------------------------------------------------------------------------
		// Error step
		// -----------------------------------------------------------------------------------------------------------
		NET_ERROR:
			// Reset commands
			NET.PAR.enable_connect := FALSE;
			NET.CMD.connect := FALSE;

			// Get more error information
			IF(NET.ERR.no = 0) THEN
				NET.ERR.no := FileIoGetSysError();
			END_IF
			NET.ERR.active := TRUE;
			IF(NET.ERR.no=26228) THEN
				brsstrcpy(ADR(NET.ERR.text), ADR('connection rejected: check network protocol, username and password'));
			ELSIF(DevLink_0.status = fiERR_DEVICE_ALREADY_EXIST) THEN
				brsstrcpy(ADR(NET.ERR.text), ADR('device is already connected'));
			END_IF

			// Reset error
			IF(NET.CMD.error_reset) THEN
				NET.CMD.error_reset := FALSE;
				NET.ERR.active := FALSE;
				NET.ERR.no := 0;
				brsmemset(ADR(NET.ERR), 0, SIZEOF(NET.ERR));
				NET.PAR.state_machine := NET_WAIT;
			END_IF
	END_CASE;

END_PROGRAM

PROGRAM _EXIT
	REPEAT
		DevUnlink_0.enable := 1;
		DevUnlink_0.handle := DevLink_0.handle;
		DevUnlink_0;
		UNTIL DevUnlink_0.status <> ERR_FUB_BUSY
	END_REPEAT;
END_PROGRAM
```

### Program Logical/Test (IEC)

#### Variables.var
```iecst
VAR
	Var1 : USINT;
END_VAR
```

#### Main.st
```iecst
PROGRAM _INIT

END_PROGRAM

PROGRAM _CYCLIC
	Var1 := Var1 + 1;

END_PROGRAM
```

Listed in the project but not available here: Logical/Global.typ, Logical/Global.var, Logical/USBdevice
